// TwinCAT 3 PLC project PLC1
// ProgramVersion: 3.1.4023.0
// libraries:
//   Tc2_Standard, * (Beckhoff Automation GmbH)
//   Tc2_System, * (Beckhoff Automation GmbH)
//   Tc2_Utilities, * (Beckhoff Automation GmbH)
//   Tc3_Module, * (Beckhoff Automation GmbH)
// project tree:
//   / PlcTask.TcTTO
//   POUs/ MAIN.TcPOU
//   Xls_Logger/DUT/ ST_CsvTableRowData.TcDUT, ST_Record.TcDUT
//   Xls_Logger/ FB_Xls_Logger.TcPOU

CONFIGURATION PLC1
    RESOURCE PLC ON TwinCAT3
        TASK PlcTask(INTERVAL := T#1ms, PRIORITY := 20);
        PROGRAM MAIN WITH PlcTask : MAIN;
    END_RESOURCE
END_CONFIGURATION

// ---- Xls_Logger/DUT/ST_CsvTableRowData.TcDUT
TYPE ST_CsvTableRowData :
STRUCT
	sTimeStamp:STRING;
	sDescription:STRING;
	sValue:STRING;
	sUnit:STRING;
END_STRUCT
END_TYPE

// ---- Xls_Logger/DUT/ST_Record.TcDUT
TYPE ST_Record :
STRUCT
	bEnableRecord:BOOL:=TRUE;
	sDescription:STRING:='Data..';
	rVal:REAL;
END_STRUCT
END_TYPE

// ---- POUs/MAIN.TcPOU
PROGRAM MAIN
VAR
	//Logger FB
	fbXls_Logger:FB_Xls_Logger;
	bStartStopLog:BOOL;
	sFilePath:STRING:='C:\Temp\';  //
	sFileName:STRING:='Records';
	sJobName:STRING:='Job1';
	
	//Data to recored
	arrRecordsData:ARRAY[1..main.fbXls_Logger.iMaxRecords]OF ST_Record;
	
	
	//analog parameter simulator
	tonGenerator:ton;
	randomNumber:drand;
	i: INT;
	bEnable: BOOL:=TRUE;
	
	
	
END_VAR


//-------create analog random values ( for testing the logger )-------
tonGenerator(IN:= NOT tonGenerator.Q , PT:=T#1MS , Q=> , ET=> );
IF tonGenerator.Q AND bEnable THEN
	FOR i:=1 TO main.fbXls_Logger.iMaxRecords DO
		IF arrRecordsData[i].bEnableRecord THEN
			randomNumber();
			arrRecordsData[i].rVal:=randomNumber.Num*100;
			arrRecordsData[i].sDescription:=concat('Data ',INT_TO_STRING(i));
		END_IF	
	END_FOR
ELSIF tonGenerator.Q then
	FOR i:=1 TO main.fbXls_Logger.iMaxRecords DO
			arrRecordsData[i].rVal:=i;
			arrRecordsData[i].sDescription:=concat('Data ',INT_TO_STRING(i));	
	END_FOR
END_IF
//-----End analog Simulator code----------------------------------------



//Call Logger FB
fbXls_Logger(bLog:=bStartStopLog,
			 sFilePath:=sFilePath,
			 sFileName:=sFileName,
			 sJobName:=sJobName,
			 arrRecordsData:=arrRecordsData
			);

END_PROGRAM

// ---- Xls_Logger/FB_Xls_Logger.TcPOU
FUNCTION_BLOCK FB_Xls_Logger
VAR_INPUT
	bLog:BOOL;//TRUE = start logging, FALSE = Stop logging
	eLogMode:(TIMER_INTERVAL,TASK_CYCLE_TIME);
	iloggingRateSec:DINT:=1; // sampling rate in secounds
	sFilePath:STRING:='C:\Temp\';
	sFileName:STRING:='Records';
	sJobName:STRING:='Job1';
	arrRecordsData:ARRAY[1..iMaxRecords]OF ST_Record;
	
END_VAR
VAR_OUTPUT
	iCurretBufferLoad:DINT;
	sStartRecoredTime:STRING;
	sEndRecoredTime:STRING;
	sCurrentSystemTime:STRING;
	sCurrentSystemDate:STRING;
	sCustomTimeStamp:STRING;
	bFileError:BOOL;
END_VAR
VAR
	arrBuffer:ARRAY[1..iMaxBufferSize]OF STRING(255);
	sRecordLine:STRING(255);
	sBufferToWrite:STRING(255*iMaxBufferSize);
	iBufferToWriteSize:UDINT:=0;
	rTrig_StartLog:r_trig;
	fTrig_EndLog:f_trig;
	fbLocalSystemTime:FB_LocalSystemTime;
	sFileHeader:STRING(255);
	i: UDINT;
	iActualBufferRecoreds:UDINT;
	
	fbFileOpen					:	FB_FileOpen;
	fbFileClose					:	FB_FileClose;
	fbFileWrite					:	FB_FileWrite;
	fbFileGet					:	FB_FileGets;
	fbFileRename				:	FB_FileRename;
	
	bWrite:BOOL:=FALSE;
	eFileWriteState:(INIT,OpenFile,WriteToFile,CloseFile,ERROR);
	rtrigWriteToFile:r_trig;
	tonRecPulse:ton;
	
	sRowToWrite: STRING(255);
	bFillBuffer: BOOL;
END_VAR
VAR CONSTANT
	iMaxBufferSize:UDINT:=70; //record buffer size
	iMaxRecords:INT:=10;// max recording parameters 
	//iMaxReadRecords:UDINT:=100000;
END_VAR

//Get system time
ACT_SystemTime();

//Start/Stop recording
rTrig_StartLog(CLK:=bLog );
fTrig_EndLog(CLK:= bLog);

//---start recording-----
IF rTrig_StartLog.Q THEN
	//set file headers
	sFileHeader:= concat(sJobName,'$nDate$TTime');
	FOR i:=1 TO iMaxRecords DO
		IF arrRecordsData[i].bEnableRecord THEN
			sFileHeader:=concat(sFileHeader,
							concat('$T',arrRecordsData[i].sDescription));
		END_IF
	END_FOR
	
	sBufferToWrite:=sFileHeader;
	iBufferToWriteSize:=LEN(sFileHeader);
	
	//set file name
	fbFileOpen.sPathName:=concat(sFilePath,
						concat(sFileName,
							concat('_',
								concat(sJobName,
									concat('_',
										concat(sCurrentSystemDate,'.xls'))))));
	

	eFileWriteState:=INIT;
	fbFileRename(sOldName:=fbFileOpen.sPathName,sNewName:=fbFileOpen.sPathName,bExecute:=TRUE);
	
END_IF

IF fbFileRename.bExecute and NOT fbFileRename.bBusy THEN
	fbFileRename.bExecute:=FALSE;
	IF fbFileRename.bError THEN
		bWrite:=TRUE;
	END_IF	
END_IF


	
// filling buffer with new line by recored reate
tonRecPulse(IN:= bLog, PT:= DINT_TO_TIME(iloggingRateSec*1000));
CASE eLogMode OF
	TIMER_INTERVAL:
		IF tonRecPulse.Q THEN
			bFillBuffer:=TRUE;	
		END_IF
		
	TASK_CYCLE_TIME:
			bFillBuffer:=TRUE;
	
END_CASE

IF bFillBuffer AND bLog THEN
	tonRecPulse(IN:= FALSE);
	bFillBuffer:=FALSE;	
	
	//create new record line
	sRecordLine:=concat('$n',
					concat(sCurrentSystemDate,
						concat('$T', sCurrentSystemTime)));
		FOR i:=1 TO iMaxRecords DO
			IF arrRecordsData[i].bEnableRecord THEN
				sRecordLine:=concat(sRecordLine,
								concat('$T',REAL_TO_STRING(arrRecordsData[i].rVal)));					
			END_IF
		END_FOR
	iActualBufferRecoreds:=Push(sRecordToPush:= sRecordLine);
END_IF

//write buffer to file
rtrigWriteToFile(CLK:=iActualBufferRecoreds > iMaxBufferSize - 10);

IF (rtrigWriteToFile.Q) OR fTrig_EndLog.Q THEN
	memset(ADR(sBufferToWrite),0,SIZEOF(sBufferToWrite));
	iBufferToWriteSize:=0;
	FOR i:=1 TO iActualBufferRecoreds DO	
		sRowToWrite:=pop();
		memcpy((ADR(sBufferToWrite)+iBufferToWriteSize),ADR(sRowToWrite),LEN(sRowToWrite));
		iBufferToWriteSize:=iBufferToWriteSize+LEN(sBufferToWrite);
	END_FOR
	bWrite:=TRUE;
END_IF


CASE eFileWriteState OF
	INIT:
		fbFileOpen(bExecute:=FALSE);
		fbFileWrite(bExecute:=FALSE);
		fbFileClose(bExecute:=FALSE);
		bFileError:=FALSE;
		IF bWrite THEN
			bWrite:=FALSE;
			eFileWriteState:=OpenFile;
		END_IF
		
	OpenFile:
		fbFileOpen(bExecute:=TRUE);
		IF NOT fbFileOpen.bBusy THEN
			IF NOT fbFileOpen.bError THEN
				eFileWriteState:=WriteToFile;
			ELSE
				bFileError:=TRUE;
				eFileWriteState:=ERROR;
			END_IF
		END_IF
		
	WriteToFile:
		fbFileWrite(hFile:= fbFileOpen.hFile, pWriteBuff:= ADR(sBufferToWrite), cbWriteLen:=iBufferToWriteSize , bExecute:= TRUE);
		IF NOT fbFileWrite.bBusy THEN
			IF NOT fbFileWrite.bError THEN
				memset(ADR(sBufferToWrite),0,SIZEOF(sBufferToWrite));
				eFileWriteState:=CloseFile;
			ELSE
				bFileError:=TRUE;
				eFileWriteState:=ERROR;
			END_IF
		END_IF
	
	CloseFile:
		fbFileClose(hFile:= fbFileOpen.hFile, bExecute:= TRUE);
		IF NOT fbFileWrite.bBusy THEN
			IF NOT fbFileWrite.bError THEN
				eFileWriteState:=INIT;
			ELSE
				bFileError:=TRUE;
				eFileWriteState:=ERROR;
			END_IF
		END_IF
		
	ERROR:
		bFileError:=TRUE;
		
END_CASE


fbFileOpen(
	nMode:= FOPEN_MODEAPPEND OR FOPEN_MODEPLUS OR FOPEN_MODETEXT, 
	ePath:= PATH_GENERIC, 
	bExecute:= , 
	tTimeout:= T#5S, 
	bBusy=> , 
	bError=> , 
	nErrId=> , 
	hFile=> );
	
fbFileWrite(
	sNetId:= , 
	hFile:= fbFileOpen.hFile, 
	pWriteBuff:= , 
	cbWriteLen:= , 
	bExecute:= , 
	tTimeout:= T#10S, 
	bBusy=> , 
	bError=> , 
	nErrId=> , 
	cbWrite=> );
	
fbFileClose(
	sNetId:= , 
	hFile:= fbFileOpen.hFile, 
	bExecute:= , 
	tTimeout:= T#10S, 
	bBusy=> , 
	bError=> , 
	nErrId=> );

fbFileRename(
	sNetId:= , 
	sOldName:= , 
	sNewName:= , 
	ePath:= PATH_GENERIC, 
	bExecute:= , 
	tTimeout:= T#5S, 
	bBusy=> , 
	bError=> , 
	nErrId=> );

ACTION ACT_SystemTime:
//read current system time
fbLocalSystemTime(bEnable:= TRUE);


//System time to strings 1. time 2. date
sCurrentSystemTime:=concat(concat(concat(concat(concat(concat(METH_TimeParToString(fbLocalSystemTime.systemTime.wHour),':'),METH_TimeParToString(fbLocalSystemTime.systemTime.wMinute)),':'),METH_TimeParToString(fbLocalSystemTime.systemTime.wSecond)),':'),WORD_TO_STRING(fbLocalSystemTime.systemTime.wMilliseconds));
sCurrentSystemDate:=concat(concat(concat(concat(METH_TimeParToString(fbLocalSystemTime.systemTime.wDay),'.'),METH_TimeParToString(fbLocalSystemTime.systemTime.wMonth)),'.'),WORD_TO_STRING(fbLocalSystemTime.systemTime.wYear));
sCustomTimeStamp:=concat(concat(sCurrentSystemDate ,' '),sCurrentSystemTime);

//Set local time
END_ACTION

METHOD METH_ConcatPtr : BOOL
VAR_INPUT
	src1Addr : POINTER TO STRING; //The address of source string 1
	src1Size : UDINT; //The size of source string 1
	src2Addr : POINTER TO STRING; //The address of source string 2
	src2Size : UDINT;//The size of source string 2
	
	destinationAddr : POINTER TO STRING; //The address of the destination string
	destinationSize : UDINT; //The size of the destination string
END_VAR
VAR_OUTPUT
	error : STRING(80); //Error message if the concat wasn't successful.
END_VAR

VAR
	i: UDINT;
	src1Len:UDINT;
END_VAR
METH_ConcatPtr := TRUE;
IF src1Size + src2Size > destinationSize THEN
	METH_ConcatPtr := FALSE;
	error := 'Destination string is not big enough';
	RETURN;
END_IF

//Check length source string 1
FOR i:=0 TO src1Size -1 DO
	IF src1Addr^[i] = 0 THEN
		src1Len:=i;
		EXIT;
	END_IF
END_FOR

//Set first source string 1 to destination
IF MEMCPY(destinationAddr, src1Addr, src1Len) = 0 THEN
	METH_ConcatPtr := FALSE;
	error := 'Incorrect parameter values. destAddr == 0 or srcAddr==0 or n == 0';//taken from beckhoff documentation.
END_IF

IF MEMCPY(destinationAddr + src1Len, src2Addr, src2Size) = 0 THEN
	METH_ConcatPtr := FALSE;
	error := 'Incorrect parameter values. destAddr == 0 or srcAddr==0 or n == 0';//taken from beckhoff documentation.
END_IF
END_METHOD

METHOD METH_TimeParToString : string
VAR_INPUT
	wTimePar:WORD;
END_VAR
IF wTimePar < 10 THEN
	METH_TimeParToString:=concat(INT_TO_STRING(0),WORD_TO_STRING(wTimePar));
ELSE
	METH_TimeParToString:=WORD_TO_STRING(wTimePar);
END_IF
END_METHOD

METHOD PUBLIC Pop : String(1000)
VAR_INPUT
END_VAR
VAR
		i: DINT;
END_VAR
Pop:=arrBuffer[1];
arrBuffer[iMaxBufferSize] := '' ;
	
FOR i:=1 TO (iMaxBufferSize) -1 DO
	arrBuffer[i]:=arrBuffer[i+1];
END_FOR
END_METHOD

METHOD PUBLIC Push : UDINT
VAR_INPUT
	sRecordToPush:STRING(1000);
END_VAR

VAR
	i: UDINT;
END_VAR
FOR i:=1 TO (iMaxBufferSize) DO
	IF arrBuffer[i]='' THEN
		arrBuffer[i]:=sRecordToPush;
		Push:=i;
		EXIT;
	END_IF
	
END_FOR
END_METHOD

END_FUNCTION_BLOCK
